KUKA KRL program: sample_program_with_globals.src, sample_program_with_globals.dat

--- sample_program_with_globals.src ---
&ACCESS RVP
&PARAM EDITMASK = *
&PARAM TEMPLATE = C:\KRC\Roboter\Template\vorgabe
DEF sample_program_with_globals( )

END

GLOBAL DEFFCT INT SampleFuncGlobal()
    return 7
ENDFCT

--- sample_program_with_globals.dat ---
&ACCESS RVP
&PARAM EDITMASK = *
&PARAM TEMPLATE = C:\KRC\Roboter\Template\vorgabe
DEFDAT sample_program_with_globals
;FOLD EXTERNAL DECLARATIONS;%{PE}%MKUKATPBASIS,%CEXT,%VCOMMON,%P
;FOLD BASISTECH EXT;%{PE}%MKUKATPBASIS,%CEXT,%VEXT,%P
EXT  BAS (BAS_COMMAND  :IN,REAL  :IN )
DECL INT SUCCESS
;ENDFOLD (BASISTECH EXT)
;FOLD USER EXT;%{E}%MKUKATPUSER,%CEXT,%VEXT,%P
;Make your modifications here
GLOBAL INT testVariableGlobal = 35
;ENDFOLD (USER EXT)
;ENDFOLD (EXTERNAL DECLARATIONS)
ENDDAT
